PROGRAM MAIN
VAR
fbTLControl			:	FB_TLControl;
fbITPControl		:	FB_ITPControl;
fbConvOpenCheck		:	FB_ConvOpen_Check;
fb_TimeStamp 		:	FB_UpdateTimeStamp;
bMsg_Init			:	BOOL := FALSE;

fbRecipe : RecipeManCommands;
recipe_name			:	STRING := 'file1';
bLog_Trigger 		:	BOOL;
Timer1				:	TON;
bFlag1				: BOOL := FALSE;
rInit	:	R_TRIG;

			
END_VAR


// ================  MISC  ================
fb_TimeStamp();
IOSignal_control();

// ================  CONVEYOR COLD START SEQUENCE  ================ 
IF IO.bStartup_State THEN							(*all hardware outputs are off*)
	IO_control.bMotor1 := FALSE;
	IO_control.bMotor2 := FALSE;
	IO_control.bMotor3 := FALSE;
	IO_control.bMotor4 := FALSE;
	
	IO_control.bGreenLight := FALSE;
	IO_control.bYellowLight := FALSE;
	IO_control.bRedLight := FALSE;
	IO_control.bBuzzer := FALSE;
	
	IF IO_control.bReset AND IO_control.bEstop OR bFlag1 THEN
		bFlag1 := TRUE;
		IO_control.bGreenLight := FALSE;
		IO_control.bYellowLight := TRUE;
		IO_control.bRedLight := FALSE;
		IO_control.bBuzzer := TRUE;
		Timer1(IN:= TRUE, PT := T#2S);
		IF Timer1.Q THEN
			IO_control.bScanner_PwrCtrl := TRUE;
			IO.bStartup_State := FALSE;
			IO.bSystem_Enabled := TRUE;
			bFlag1 := FALSE;
			Timer1(IN := FALSE);
		END_IF
	END_IF
END_IF

// one-time init when PLC starts / task enables
rInit(CLK := IO.bStartup_State);
IF rInit.Q THEN
    IO.fbClient_QR.fbRx.sPut := 'null';   // clear any leftover frame
    IO.sCam_Received_msg     := '';
    IO_Conveyor.bScan_Start  := FALSE;
    IO_Conveyor.bScan_Complete := FALSE;
    IO_Conveyor.bScan_Failed := FALSE;
    IO_Conveyor.bScan_ERROR  := FALSE;
   // IO.Cam_Timeout(IN := FALSE);             // be sure timer is reset
END_IF

// ================  CONVEYOR COLD STARTUP (TO ENABLE SYSTEM)  ================ 
Conveyor_Init() ;		(*conveyor init function*)

IF IO.bSystem_Enabled AND IO_control.bReset THEN	(*alarm pop-up for cold start*)
	IO.bSystem_Enabled := FALSE;
	IO_control.bYellowLight := FALSE;
	IO_control.bBuzzer := FALSE ;
	IO.bSystem_standby := TRUE;
END_IF

// ================  CONVEYOR OPERATION MODE SETUP  ================
IF IO.bSystem_standby THEN
	ModeEvent_Handling();		(*alarm pop-up for cold start*)
	bMsg_Init := TRUE;
	IO.bConv_Init_Cmd := IO_control.bReset OR IO.bConv_Init_Cmd;		(*operation mode logic*)
	IO.bPre_AutoMode := IO.bConv_Init_Ready AND IO_control.bEstop AND NOT IO_control.bStop  AND NOT IO_control.bManualToggle ;
	IO.bAutoMode := (IO_control.bStart OR IO.bAutoMode) AND IO.bPre_AutoMode ;
	IO.bManualMode := NOT IO.bAutoMode ;
	IO.bEstop_State := NOT IO_control.bEstop OR IO.bEstop_State ;
	
	(*tower light logic*)
	IO.fbBlinker();
	IO.fbBlinker.BlinkInterval := T#1000MS;
	fbTLControl();
END_IF

//Indicator for conv ready for operation
IF IO.bAutoMode THEN
	IO.bConv_Ready := TRUE;
	IO.fbWCS_MsgPush();
	IO.fbWCS_MsgHandler();
ELSE
	IO.bConv_Ready := FALSE ;
END_IF

// ================  ITP LOGIC  ================
fbITPControl();		

// ================  KEYENCE SCANNER  ================
IO.fbKeyence();
Scanner_PwrCtrl();

// ================  OPEN STATUS CHECKING FOR EACH CONVEYOR + CONV PROCESS  ================
IF NOT IO.bInterrupt_State THEN
	fbConvOpenCheck();
	IO.fbConv4();
	IO.fbConv3();
	IO.fbConv2();
	IO.fbConv1(); 
END_IF

// ================  CONV READY FOR OPERATON CHECKING  ================
IF IO.bAutoMode THEN
	IO.bConv_Ready := TRUE;
	IO.fbWCS_MsgPush();
	IO.fbWCS_MsgHandler();
ELSE
	IO.bConv_Ready := FALSE ;
END_IF

// ================  KUKA ROBOT  ================
ExtMode_Init();
KUKAFunction_IO();
IO.fbKUKA_Main();
KUKAData_IO();

// ================  TCP/IP COMMS  ================
(*TCP/IP Comm starter*)
IO.fbCloseAll( sSrvNetID := IO.sSrvNetID, bExecute:= IO.bInitialize );
IF IO.fbCloseAll.bBusy OR IO.fbCloseAll.bError THEN
	RETURN;
END_IF	
IO.bInitialize := FALSE;
IO.fbClient_QR( sSrvNetId := IO.sSrvNetID, bEnable := IO.bScannerEnable, bLog := IO.bLog );
IO.fbClient_ASRS( sSrvNetId := IO.sSrvNetID, bEnable := IO.bScannerEnable, bLog := IO.bLog );

//Tcp/ip Msg init to 'null'	
IF NOT bMsg_Init THEN
	IO.fbClient_ASRS.fbRx.sPut := 'null';
	IO.fbClient_QR.fbRx.sPut := 'null';
	bMsg_Init := TRUE;
END_IF

// ================  POSTMAN COMMS  ================
Postman_MAIN();
Postman_filter();
Data_Shifting();
device_rtrig();

// ================  DIGIIOT COMMS  ================
DIGI_Main();

////////logging function
////////Process_Logging();
////////MSG.ACTION_SCNR_ON := IO.Received_msg ;

END_PROGRAM

(* stored: Version 1.1.0.1, ProductVersion 3.1.4024.12
   POU MAIN: Id {acb6eb24-017d-4845-9e8d-c9c53fe62c4c}, SpecialFunc None *)
